(* LS Electric XG5000 project: 첫프로젝트 *)
(* PLC LSPLC *)
(* module base 0 slot 0: 입력 모듈:XGI-D22A/B (DC 24V 입력, 16점 (전류소스 싱크공용/ 전류소스 입력)) *)
(* module base 0 slot 1: 출력 모듈:XGQ-RY2A/B (릴레이 출력, 16점 (2A용, Varistor 없음/Varistor 부착)) *)
(* module base 0 slot 2: 출력 모듈:XGQ-RY1A (릴레이 출력, 8점 (2A용, 단독 COM.)) *)
VAR_GLOBAL
    램프1 AT %QX0.1.2 : BOOL; (* 출력입니다2 *)
END_VAR

(* Comments on direct variables
%IX0.0.0	5번포트
*)

PROGRAM NewProgram (* task: 스캔 프로그램 *)
VAR
    램프 AT %QX0.1.1 : BOOL; (* 출력입니다 *)
END_VAR
VAR_EXTERNAL
    램프1 : BOOL; (* AT %QX0.1.2 *) (* 출력입니다2 *)
END_VAR

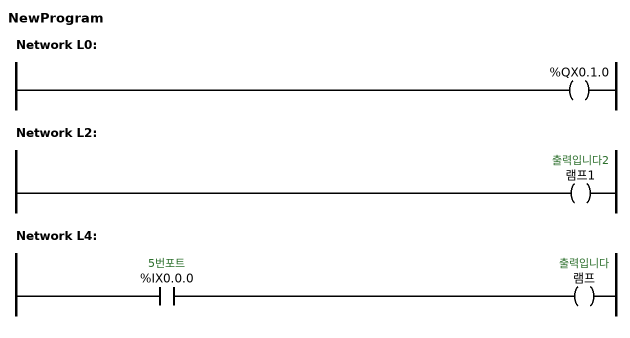
(* Rung L0 *)
%QX0.1.0 := TRUE;
(* Rung L2 *)
램프1 := TRUE;
(* Rung L4 *)
램프 := %IX0.0.0;
END_PROGRAM